VAR_GLOBAL
	instOperatingmode	:	FactoryIO.FB_OperatingMode;
	currentStateOperatingMode	:	FactoryIO.OperatingMode;
	permissionHardware	:	BOOL := TRUE;
	permissionSafety	:	BOOL := TRUE;
END_VAR

(* stored: Version 1.1.0.1
   GVL OperatingMode: Id {c6370a8f-09ee-48de-964a-204ce261ab37} *)
